TYPE ST_AxisGroupDescription :
STRUCT
	sGroupName : STRING(nMAX_AXIS_GROUP_NAME);
	iAxesInGroup : INT;
END_STRUCT
END_TYPE

(* stored: Version 1.1.0.1, ProductVersion 3.1.4024.11
   DUT ST_AxisGroupDescription: Id {38fa0151-2a96-43c9-99b3-0118e0ccb3d1} *)
